% RSLogix 500 project PROJECT_2_PROX_SENSOR_LIGHT_DETECTION.RSS, saved by version 8.30.00.16 %
PROJECT "PROX.SEN"    % processor: Bul.1763 MicroLogix 1100 Series B %

PROGRAM FILES
  LAD 2 "SYSTEM"  3 rungs
  LAD 3 "IN/OUT"  4 rungs
  LAD 4 "MAIN"  6 rungs

DATA FILES
  O0 OUTPUT  4 elements
  I1 INPUT  6 elements
  S2 STATUS  66 elements
  B3 BINARY  100 elements
  T4 TIMER  10 elements
  C5 COUNTER  10 elements
  R6 CONTROL  1 elements
  N7 INTEGER  10 elements
  F8 FLOAT  1 elements

LADDER 2 "SYSTEM"
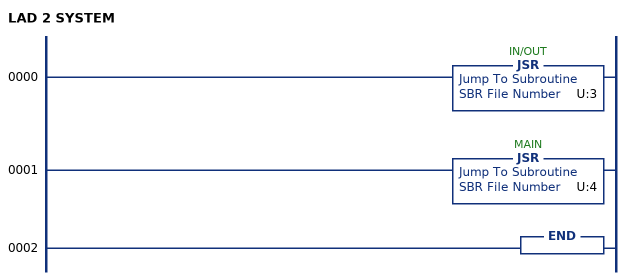
% Rung: 0 %
SOR JSR U:3 EOR
%   U:3  "IN/OUT" %
% Rung: 1 %
SOR JSR U:4 EOR
%   U:4  "MAIN" %
% Rung: 2 %
SOR END EOR

LADDER 3 "IN/OUT"
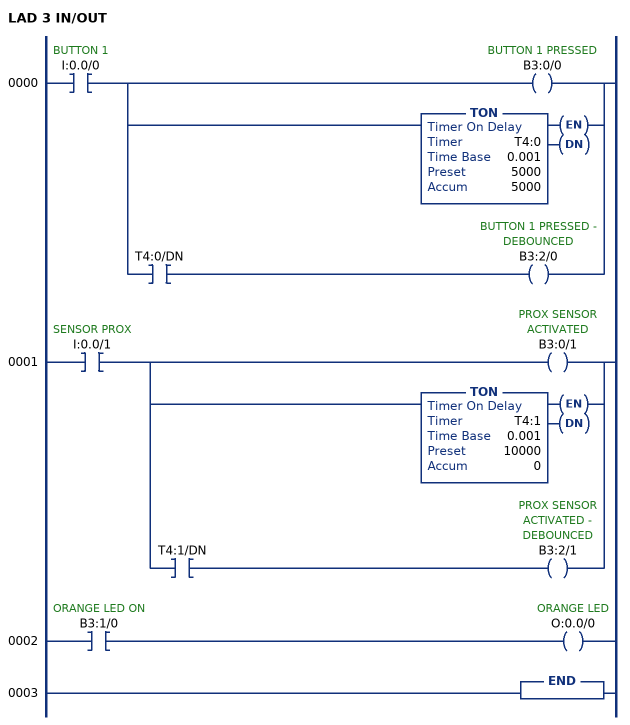
% Rung: 0 %
SOR XIC I:0.0/0 BST OTE B3:0/0 NXB BST TON T4:0 0.001 5000 5000 NXB XIC T4:0/DN OTE B3:2/0 BND BND EOR
%   I:0.0/0  "BUTTON 1" %
%   B3:0/0  "BUTTON 1 PRESSED" %
%   B3:2/0  "BUTTON 1 PRESSED - DEBOUNCED" %
% Rung: 1 %
SOR XIC I:0.0/1 BST OTE B3:0/1 NXB BST TON T4:1 0.001 10000 0 NXB XIC T4:1/DN OTE B3:2/1 BND BND EOR
%   I:0.0/1  "SENSOR PROX" %
%   B3:0/1  "PROX SENSOR ACTIVATED" %
%   B3:2/1  "PROX SENSOR ACTIVATED - DEBOUNCED" %
% Rung: 2 %
SOR XIC B3:1/0 OTE O:0.0/0 EOR
%   B3:1/0  "ORANGE LED ON" %
%   O:0.0/0  "ORANGE LED" %
% Rung: 3 %
SOR END EOR

LADDER 4 "MAIN"
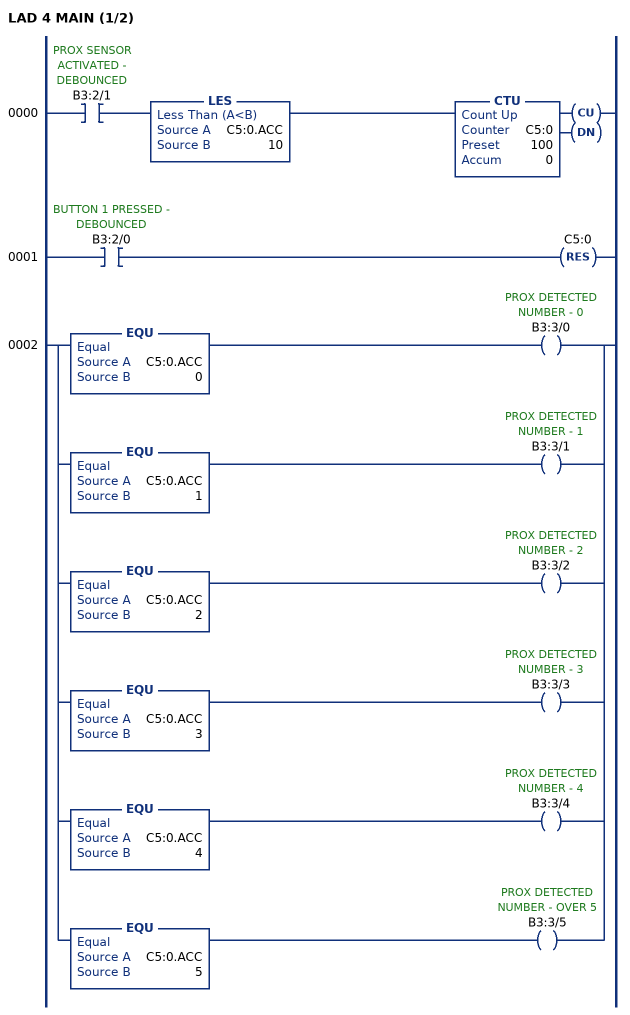
% Rung: 0 %
SOR XIC B3:2/1 LES C5:0.ACC 10 CTU C5:0 100 0 EOR
%   B3:2/1  "PROX SENSOR ACTIVATED - DEBOUNCED" %
% Rung: 1 %
SOR XIC B3:2/0 RES C5:0 EOR
%   B3:2/0  "BUTTON 1 PRESSED - DEBOUNCED" %
% Rung: 2 %
SOR BST EQU C5:0.ACC 0 OTE B3:3/0 NXB EQU C5:0.ACC 1 OTE B3:3/1 NXB EQU C5:0.ACC 2 OTE B3:3/2 NXB EQU C5:0.ACC 3 OTE B3:3/3 NXB EQU C5:0.ACC 4 OTE B3:3/4 NXB EQU C5:0.ACC 5 OTE B3:3/5 BND EOR
%   B3:3/0  "PROX DETECTED NUMBER - 0" %
%   B3:3/1  "PROX DETECTED NUMBER - 1" %
%   B3:3/2  "PROX DETECTED NUMBER - 2" %
%   B3:3/3  "PROX DETECTED NUMBER - 3" %
%   B3:3/4  "PROX DETECTED NUMBER - 4" %
%   B3:3/5  "PROX DETECTED NUMBER - OVER 5" %

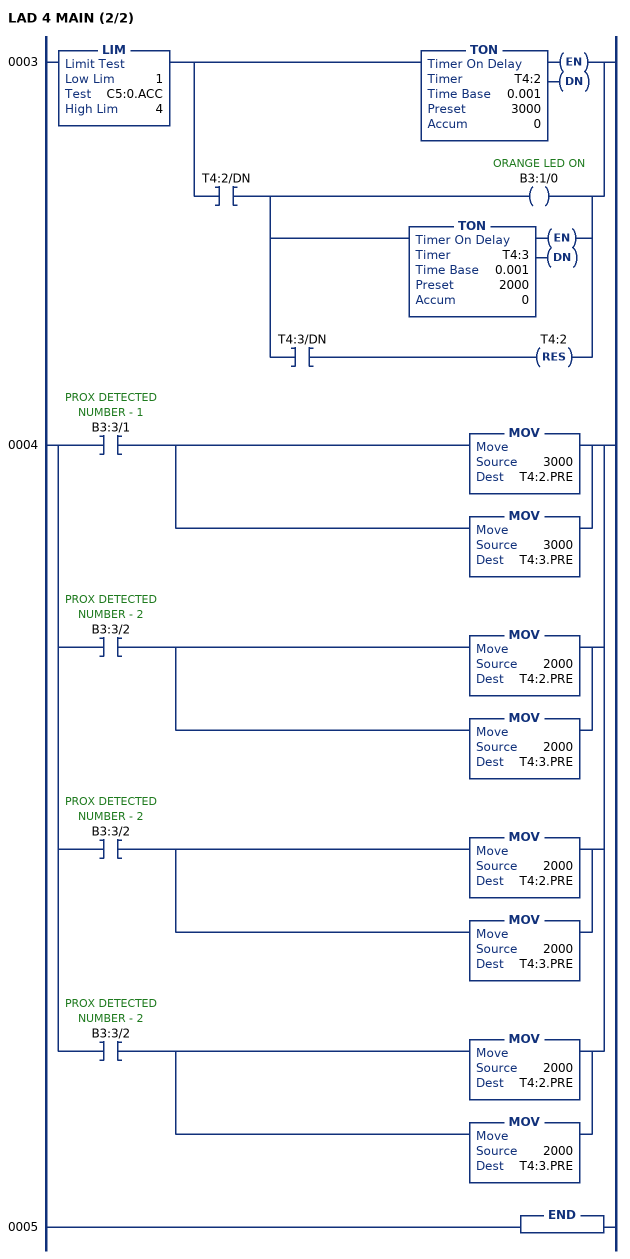
% Rung: 3 %
SOR LIM 1 C5:0.ACC 4 BST TON T4:2 0.001 3000 0 NXB XIC T4:2/DN BST OTE B3:1/0 NXB TON T4:3 0.001 2000 0 NXB XIC T4:3/DN RES T4:2 BND BND EOR
%   B3:1/0  "ORANGE LED ON" %
% Rung: 4 %
SOR BST XIC B3:3/1 BST MOV 3000 T4:2.PRE NXB MOV 3000 T4:3.PRE BND NXB XIC B3:3/2 BST MOV 2000 T4:2.PRE NXB MOV 2000 T4:3.PRE BND NXB XIC B3:3/2 BST MOV 2000 T4:2.PRE NXB MOV 2000 T4:3.PRE BND NXB XIC B3:3/2 BST MOV 2000 T4:2.PRE NXB MOV 2000 T4:3.PRE BND BND EOR
%   B3:3/1  "PROX DETECTED NUMBER - 1" %
%   B3:3/2  "PROX DETECTED NUMBER - 2" %
% Rung: 5 %
SOR END EOR

OTHER DOCUMENTED ADDRESSES
  ORANGE_LED  
  U3  

DATA TABLE (non-zero values as saved)
DATA B3
% B3:0 % 0X0001 0X0000 0X0001 0X0001 0X0000 0X0000 0X0000 0X0000 0X0000 0X0000
DATA T4
% .PRE .ACC %
% T4:0 % 5000 5000
% T4:1 % 10000 0
% T4:2 % 3000 0
% T4:3 % 2000 0
DATA C5
% .PRE .ACC %
% C5:0 % 100 0
